FUNCTION Convert_LREAL_TO_BYTE : BOOL
VAR_INPUT
	in : LREAL;
	out : REFERENCE TO BYTE;
END_VAR
VAR
	converted : BYTE;
END_VAR

converted := LREAL_TO_BYTE(in);

IF (BYTE_TO_LREAL(converted) <> in) THEN
	RETURN;
END_IF

out := converted;
Convert_LREAL_TO_BYTE := TRUE;

END_FUNCTION

(* stored: Version 1.1.0.1, ProductVersion 3.1.4024.12
   POU Convert_LREAL_TO_BYTE: Id {f25f8a48-8e76-46de-97ea-352ab91936d8}, SpecialFunc None *)
